# EPICS alarm handler configuration: example.alhConfig
GROUP NULL TOP
$ALIAS Alarms

CHANNEL TOP numberbox
